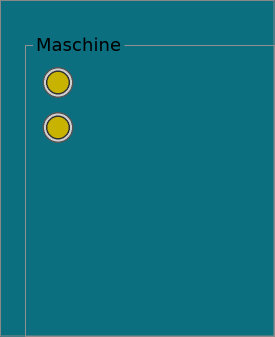
VISUALIZATION Visualization  // 275x337
    GroupBox (25,37 250x300), "Maschine"
        Lamp1 (13,28 40x35), style: Lamp-Lamp1-Yellow
        Lamp1 (13,73 40x35), style: Lamp-Lamp1-Yellow
END_VISUALIZATION

(* stored: Version 1.1.0.1, ProductVersion 3.1.4026.18
   Visu Visualization: Id {41bb52dc-3ba4-40b2-80e4-ac4579fbf1a3} *)
